// TwinCAT 3 PLC project Untitled1
// ProgramVersion: 3.1.4024.0
// libraries:
//   Tc2_MC2, * (Beckhoff Automation GmbH)
//   Tc2_Standard, * (Beckhoff Automation GmbH)
//   Tc2_System, * (Beckhoff Automation GmbH)
//   Tc3_Mc3PlanarMotion, * (Beckhoff Automation GmbH)
//   Tc3_Module, * (Beckhoff Automation GmbH)
//   Tc3_Physics, * (Beckhoff Automation GmbH)
// project tree:
//   DUTs/ Command.TcDUT
//   / GlobalTextList.TcGTLO, PlcTask.TcTTO, Visualization Manager.TcVMO (not stored)
//   GVLs/ GVL.TcGVL
//   POUs/ ControllerMode.TcPOU (not stored), FB_TcJoy.TcPOU, MAIN.TcPOU
//   VISUs/ Visualization.TcVIS
// real-time tasks:
//   TASK PlcTask: cycle T#10ms, priority 20, ADS port 350
//   TASK XPlanar Task3: cycle T#250us, priority 1, ADS port 351
//   TASK MC-Task (MET): cycle T#2ms, priority 2, ADS port 352
//   TASK MC-Task (MPT): cycle T#10ms, priority 3, ADS port 353
//   TASK Job Task: cycle default, priority 4
// motion (NC):
//   TASK NC-Task 1 SAF: cycle T#2ms, priority 5, ADS port 501
//   TASK NC-Task 1 SVB: cycle T#10ms, priority 9, ADS port 511
//   AXIS M1_X (id 1)
//     OtherSettings: AllowMotionCmdToSlave=true
//     encoder EncType=1
//     drive DrvType=5
//       Analog: TorqueSetpointScale=10, ScaleFactorActTorque=0.1
//       TimeComp: TaskDelayCycles=1
//     controller CtrType=1
//       CtrPara: PriorControlFactor=1
//         Observer: BandWidth=20
//   AXIS M1_Y (id 2)
//     OtherSettings: AllowMotionCmdToSlave=true
//     encoder EncType=1
//     drive DrvType=5
//       Analog: TorqueSetpointScale=10, ScaleFactorActTorque=0.1
//       TimeComp: TaskDelayCycles=1
//     controller CtrType=1
//       CtrPara: PriorControlFactor=1
//         Observer: BandWidth=20
//   AXIS M1_Z (id 3)
//     OtherSettings: AllowMotionCmdToSlave=true
//     encoder EncType=1
//     drive DrvType=5
//       Analog: TorqueSetpointScale=10, ScaleFactorActTorque=0.1
//       TimeComp: TaskDelayCycles=1
//     controller CtrType=1
//       CtrPara: PriorControlFactor=1
//         Observer: BandWidth=20
//   AXIS M1_A (id 4)
//     General: UnitName=°
//     OtherSettings: AllowMotionCmdToSlave=true
//     encoder EncType=1
//     drive DrvType=5
//       Analog: TorqueSetpointScale=10, ScaleFactorActTorque=0.1
//       TimeComp: TaskDelayCycles=1
//     controller CtrType=1
//       CtrPara: PriorControlFactor=1
//         Observer: BandWidth=20
//   AXIS M1_B (id 5)
//     General: UnitName=°
//     OtherSettings: AllowMotionCmdToSlave=true
//     encoder EncType=1
//     drive DrvType=5
//       Analog: TorqueSetpointScale=10, ScaleFactorActTorque=0.1
//       TimeComp: TaskDelayCycles=1
//     controller CtrType=1
//       CtrPara: PriorControlFactor=1
//         Observer: BandWidth=20
//   AXIS M1_C (id 6)
//     General: UnitName=°
//     OtherSettings: AllowMotionCmdToSlave=true
//     encoder EncType=1
//     drive DrvType=5
//       Analog: TorqueSetpointScale=10, ScaleFactorActTorque=0.1
//       TimeComp: TaskDelayCycles=1
//     controller CtrType=1
//       CtrPara: PriorControlFactor=1
//         Observer: BandWidth=20
// variable links:
//   XPlanar MC Project/Axes/Mover4330_1 <-> TcCOM Objects/XPlanar/Mover4330_1
//     IoToMc/STD <-> OutputsToNC3/HWToNC3
//     McToIo/STD <-> InputsFromNC3/NC3ToHW
//   Untitled1/Untitled1 Instance <-> NC-Task 1 SAF/Axes/M1_A
//     PlcTask Inputs/MAIN.fbM1_Axis[4].NcToPlc <-> Outputs/ToPlc
//     PlcTask Outputs/MAIN.fbM1_Axis[4].PlcToNc <-> Inputs/FromPlc
//   Untitled1/Untitled1 Instance <-> NC-Task 1 SAF/Axes/M1_B
//     PlcTask Inputs/MAIN.fbM1_Axis[5].NcToPlc <-> Outputs/ToPlc
//     PlcTask Outputs/MAIN.fbM1_Axis[5].PlcToNc <-> Inputs/FromPlc
//   Untitled1/Untitled1 Instance <-> NC-Task 1 SAF/Axes/M1_C
//     PlcTask Inputs/MAIN.fbM1_Axis[6].NcToPlc <-> Outputs/ToPlc
//     PlcTask Outputs/MAIN.fbM1_Axis[6].PlcToNc <-> Inputs/FromPlc
//   Untitled1/Untitled1 Instance <-> NC-Task 1 SAF/Axes/M1_X
//     PlcTask Inputs/MAIN.fbM1_Axis[1].NcToPlc <-> Outputs/ToPlc
//     PlcTask Outputs/MAIN.fbM1_Axis[1].PlcToNc <-> Inputs/FromPlc
//   Untitled1/Untitled1 Instance <-> NC-Task 1 SAF/Axes/M1_Y
//     PlcTask Inputs/MAIN.fbM1_Axis[2].NcToPlc <-> Outputs/ToPlc
//     PlcTask Outputs/MAIN.fbM1_Axis[2].PlcToNc <-> Inputs/FromPlc
//   Untitled1/Untitled1 Instance <-> NC-Task 1 SAF/Axes/M1_Z
//     PlcTask Inputs/MAIN.fbM1_Axis[3].NcToPlc <-> Outputs/ToPlc
//     PlcTask Outputs/MAIN.fbM1_Axis[3].PlcToNc <-> Inputs/FromPlc
//   Untitled1/Untitled1 Instance <-> XPlanar MC Project/Axes/Mover4330_1
//     PlcTask Inputs/MAIN.fbMover.MCTOPLC/ACT <-> McToPlc/ACT
//     PlcTask Inputs/MAIN.fbMover.MCTOPLC/COORDMODE <-> McToPlc/COORDMODE
//     PlcTask Inputs/MAIN.fbMover.MCTOPLC/SET <-> McToPlc/SET
//     PlcTask Inputs/MAIN.fbMover.MCTOPLC/SETONTRACK <-> McToPlc/SETONTRACK
//     PlcTask Inputs/MAIN.fbMover.MCTOPLC/STD <-> McToPlc/STD
//     PlcTask Outputs/MAIN.fbMover.PLCTOMC/STD <-> PlcToMc/STD

CONFIGURATION Untitled1
    RESOURCE PLC ON TwinCAT3
        TASK PlcTask(INTERVAL := T#10ms, PRIORITY := 20);
        PROGRAM MAIN WITH PlcTask : MAIN;
    END_RESOURCE
END_CONFIGURATION

// ---- DUTs/Command.TcDUT
{attribute 'qualified_only'}
{attribute 'strict'}
TYPE Command :
(
	None := 0
	,Pad	 		:= 1
	,RightStick		:= 2
	,LeftStick		:= 3
	,A				:= 4
	,B				:= 5
	,X				:= 6
	,Y				:= 7
	,L1				:= 8
	,R1				:= 9
	,L2				:= 10
	,R2				:= 11
	,Start			:= 12
	,Back			:= 13
);
END_TYPE

// ---- GVLs/GVL.TcGVL
//{attribute 'qualified_only'}
VAR_GLOBAL
	g_fbTcJoy						: FB_TcJoy;
	g_lrDeadZone					: LREAL := 10000;	
END_VAR

VAR_GLOBAL CONSTANT
	gc_lrMax_Stick					: LREAL := 32767; 
	gc_lrMax_L2R2					: LREAL := 255;
	gc_alrLowCondition_Pos			: ARRAY [0..3] OF LREAL := [100, 1000, 1000, 10000];
	gc_alrHighCondition_Pos			: ARRAY [0..3] OF LREAL := [500, 5000, 5000, 50000];
	gc_alrLowCondition_Angle		: ARRAY [0..3] OF LREAL := [100, 1000, 1000, 10000];
END_VAR

// ---- POUs/MAIN.TcPOU
PROGRAM MAIN
VAR
	fbMover				: MC_PlanarMover;
	fbM1_Axis			: ARRAY [1..6] OF AXIS_REF;
	iMode				: INT;
END_VAR

GVL.g_fbTcJoy();

CASE iMode OF
	0: 
	ControllerMode(
		fbMover:= fbMover, 
		fbMover_Axis:= fbM1_Axis);
END_CASE

fbMover.Update();

END_PROGRAM

// ---- POUs/FB_TcJoy.TcPOU
FUNCTION_BLOCK FB_TcJoy
VAR_INPUT
END_VAR
VAR_OUTPUT
	bIsActive : BOOL;  // Are we running?
	// Controller Outputs for use in programs:
	Start_Button : BOOL; 
	Back_Button : BOOL;
	A_Button : BOOL;
	B_Button : BOOL;
	X_Button : BOOL;
	Y_Button : BOOL;
	LeftShoulder_Button : BOOL;
	RightShoulder_Button : BOOL;
	LeftStick_Button : BOOL;
	RightStick_Button : BOOL;
	DPad_Up_Button : BOOL;
	DPad_Left_Button : BOOL;
	DPad_Right_Button : BOOL;
	DPad_Down_Button : BOOL;
	iLeftStick_X_Axis : DINT;
	iLeftStick_Y_Axis : DINT;
	iRightStick_X_Axis : DINT;
	iRightStick_Y_Axis : DINT;
	iLeftTrigger_Axis : DINT;
	iRightTrigger_Axis  : DINT;
	sBatteryInfo		: STRING;
END_VAR
VAR
	// From VB App To PLC
	bHeartBeatToggle : BOOL;  // From VB App
	iADSWatchdogMS : DINT;    // If Rate is > this, all outputs go to 0.
	iADSWatchdogDeadDurationMS : DINT;    // If watchdog trips, outputs go to 0 for this long.
	bWatchdogFailureActive			: BOOL;
	bControlerInputsMustBeReleased  : BOOL;  // Are controller inputs holding us in latency lock down?
	// From PLC To VB (Status)
	iUpdateRateMS : DINT;    // Rate in MS between heartbeat changes detected.
	
	// Internal Use Only
	HeartBeatChanged_RTRIG : R_TRIG;
	bHeartBeatToggle_Last : BOOL;
	UpdateRate_TMR : TON;
	
	LatencyWatchdog_TMR : TON; // Watch for missing ADS and kill joy output for a while.
	LatencyWatchdogDeadDuration_TMR : TON; // Watchdog will kill the outputs for this long...
	
	iScanCount: DINT; // Scan counter for VB Status.
	
	bControllerConnected : BOOL;  // Is there a controller connected?
	
END_VAR

iScanCount := iScanCount+1;

UpdateRate_TMR(PT:=T#999M);

HeartBeatChanged_RTRIG(clk := bHeartBeatToggle <> bHeartBeatToggle_Last);

// VB "Just" changed heartbeat.
IF HeartBeatChanged_RTRIG.Q THEN
	bHeartBeatToggle_Last := bHeartBeatToggle;
	iUpdateRateMS := TIME_TO_DINT(UpdateRate_TMR.ET); // Grab Elapsed Time
	UpdateRate_TMR(IN:=FALSE); // Reset Timer
	UpdateRate_TMR(IN:=TRUE); // Reset Timer
END_IF

LatencyWatchdog_TMR(IN:=bHeartBeatToggle, PT:=DINT_TO_TIME(iADSWatchdogMS));

// AHH Latency Elapsed!
IF LatencyWatchdog_TMR.Q THEN
	bWatchdogFailureActive := TRUE;
	bControllerConnected := FALSE;
END_IF



//Force User to release all buttons/sticks on controller before allowing outputs again.
IF bWatchdogFailureActive AND (Start_Button OR 
	Back_Button OR 
	A_Button OR 
	B_Button OR 
	X_Button OR 
	Y_Button OR 
	LeftShoulder_Button OR 
	RightShoulder_Button OR 
	LeftStick_Button OR
	RightStick_Button OR
	DPad_Up_Button OR 
	DPad_Left_Button OR 
	DPad_Right_Button OR 
	DPad_Down_Button OR 
	iLeftStick_X_Axis <> 0 OR
	iLeftStick_Y_Axis <> 0 OR
	iRightStick_X_Axis <> 0 OR
	iRightStick_Y_Axis <> 0 OR
	iLeftTrigger_Axis <> 0 OR
	iRightTrigger_Axis <> 0)	THEN
		bControlerInputsMustBeReleased := TRUE;
ELSE
		bControlerInputsMustBeReleased := FALSE;
END_IF

LatencyWatchdogDeadDuration_TMR(IN:=bWatchdogFailureActive AND NOT bControlerInputsMustBeReleased AND bControllerConnected, PT:=DINT_TO_TIME(iADSWatchdogDeadDurationMS));

// ReEnable after setting duration expires
IF LatencyWatchdogDeadDuration_TMR.Q THEN
	bWatchdogFailureActive := FALSE;
END_IF

// Null the outputs on WD Active so we don't jog into a wall if we lose connection.
IF (bWatchdogFailureActive OR NOT bControllerConnected OR bControlerInputsMustBeReleased) THEN
		// Null all outputs now.
		Start_Button := FALSE; 
		Back_Button := FALSE; 
		A_Button := FALSE; 
		B_Button := FALSE; 
		X_Button := FALSE; 
		Y_Button := FALSE; 
		LeftShoulder_Button := FALSE; 
		RightShoulder_Button := FALSE; 
		LeftStick_Button := FALSE; 
		RightStick_Button := FALSE; 
		DPad_Up_Button := FALSE; 
		DPad_Left_Button := FALSE; 
		DPad_Right_Button := FALSE; 
		DPad_Down_Button := FALSE; 
		iLeftStick_X_Axis := 0;
		iLeftStick_Y_Axis := 0;
		iRightStick_X_Axis := 0;
		iRightStick_Y_Axis := 0;
		iLeftTrigger_Axis := 0;
		iRightTrigger_Axis := 0;
		sBatteryInfo		:= 'Unkn';
		
		UpdateRate_TMR(IN:=FALSE); // Reset Rate Timer
ELSE
	; // All is well, VB will update our values constantly.
END_IF

bIsActive := NOT bWatchdogFailureActive AND bControllerConnected AND NOT bControlerInputsMustBeReleased;

END_FUNCTION_BLOCK

// ---- VISUs/Visualization.TcVIS
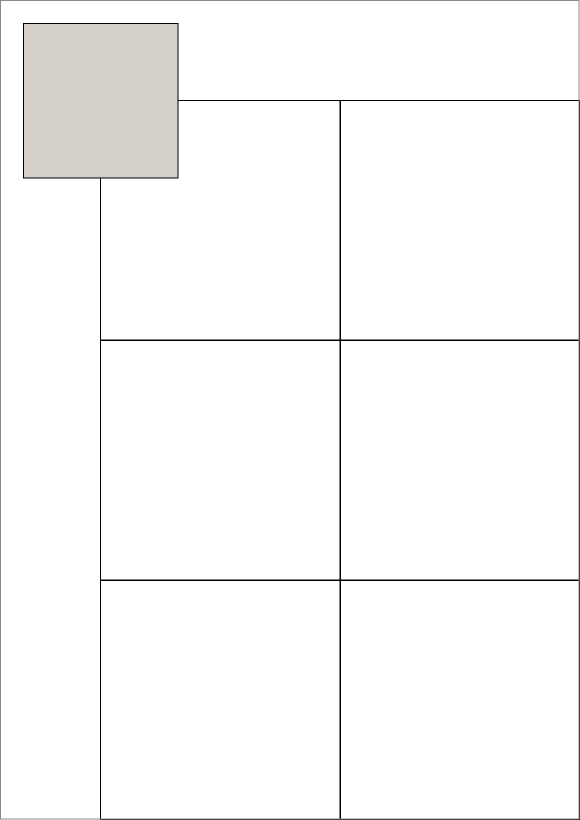
VISUALIZATION Visualization  // 580x820
    Rectangle (100,100 240x240)
    Rectangle (340,100 240x240)
    Rectangle (100,340 240x240)
    Rectangle (340,340 240x240)
    Rectangle (100,580 240x240)
    Rectangle (340,580 240x240)
    RoundedRectangle (23,23 155x155)
END_VISUALIZATION
